{attribute 'OPC.UA.DA' := '0'}
TYPE WaferPresenceSensor :
STRUCT
	Name : STRING;
	Diameter : UINT;
	InputWaferPresence AT %I* : BOOL;
END_STRUCT
END_TYPE

(* stored: Version 1.1.0.1, ProductVersion 3.1.4024.12
   DUT WaferPresenceSensor: Id {3561d092-b030-4a52-a80d-bd5d6aa27526} *)
